Fanuc KAREL source: NC0063.compact.KL

PROGRAM NC0063
%STACKSIZE=65535
%PRIORITY=65535
%NOLOCKGROUP
ROUTINE R FROM NC0063
ROUTINE R
VAR
S1 : INTEGER
S2 : INTEGER
S3 : INTEGER
BEGIN
S1=1
FOR S2=1 TO 2 DO
FOR S3=1 TO 2 DO
S1=(S1 + 1)
ENDFOR
ENDFOR
END R
BEGIN
R
END NC0063
